PROGRAM prg_TweeSignalen
VAR
	S01, S02		AT		%I*		:BOOL; 
	Q01, Q02		AT		%Q*		:BOOL;
END_VAR

Q01 := NOT(S02);
Q02 := NOT(S01);

END_PROGRAM

(* stored: Version 1.1.0.1, ProductVersion 3.1.4024.15
   POU prg_TweeSignalen: Id {d9a584fe-b010-4267-91fb-b83ff1bd3263}, SpecialFunc None *)
